PROGRAM Main
VAR
	sVersion: STRING:='1.0.0';
	M1:FB_DriveVirtual;
	M1Link:FB_NcAxis;
	bLimitFwd AT %I*: BOOL;
	bLimitBwd AT %I*: BOOL;
	bHomeSensor AT %I*: BOOL;
	bOutput1 AT %Q*: BOOL:= TRUE;
	bOutput2 AT %Q*: BOOL:= TRUE;
	bOutput3 AT %Q*: BOOL:= TRUE;
	bOutput4 AT %Q*: BOOL:= TRUE;
	bOutput5 AT %Q*: BOOL:= TRUE;
	bOutput6 AT %Q*: BOOL:= TRUE;
	bOutput7 AT %Q*: BOOL:= TRUE;
	bOutput8 AT %Q*: BOOL:= TRUE;	
	fAmplitude:LREAL:=1;
	fTest: LREAL:=0;
	iTest: INT:=0;
	bTest: BYTE:=0;
	sTest: STRING:= 'Hope it works!';
	fTestArray: ARRAY [0..99] OF LREAL;
	iIndex:INT:=0;
	iTestError:INT:=0;
	
END_VAR


//CALL ACTION TO EXECUTE FB_DriveVirtual
act();

//Update variables
iTest:=iTest+1;
fTest:=fAmplitude*SIN(iTest*2*pi/360);
bTest:=bTest+1;
iIndex:=iIndex+1;

IF iIndex>99 THEN
	iIndex:=0;
END_IF
//Make memmove to get continious signal!
MEMMOVE(destAddr:=ADR(fTestArray[0]),srcAddr:=ADR(fTestArray[1]),n:=99*8);
fTestArray[99]:=fTest;

ACTION ACT:
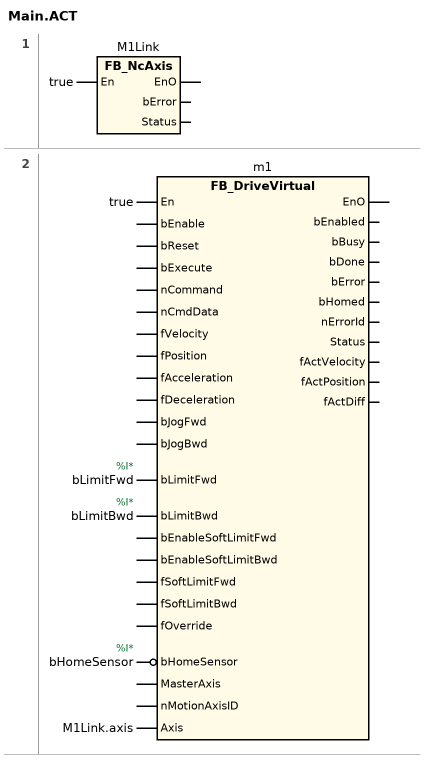
// NETWORK 1
M1Link(En := true); // FB_NcAxis

// NETWORK 2
//   bLimitFwd: AT %I*
//   bLimitBwd: AT %I*
//   bHomeSensor: AT %I*
m1(
    En := true,
    bLimitFwd := bLimitFwd,
    bLimitBwd := bLimitBwd,
    bHomeSensor := NOT bHomeSensor,
    Axis := M1Link.axis); // FB_DriveVirtual
END_ACTION

END_PROGRAM

(* stored: Version 1.1.0.1, ProductVersion 3.1.0.36
   POU Main: Id {68d5c4cd-ed5a-46ef-a7cd-a34a6aaecb11}, SpecialFunc None
   Action ACT: Id {d90d5e50-7562-49a7-958d-fc203dcb8912} *)
